// TIA Portal project "ProjectMurr-55510-en" (V18)

(* hardware
DEVICE "S7-1200 station_1"  S7-1200 Station
   slot 0: "Rack_0"  S7-1200 Rack  Rack  V1.0
   slot 1: "PLC_1"  CPU 1212FC DC/DC/DC  6ES7 212-1AF40-0XB0  V4.6
DEVICE "GSD device_1"  GSD.Device.PN
   slot 0: "Rack"  Rack  V1.0
   slot 0: "FIO"  FIO
   slot 0: "IOL_I/O_08/08 + PQI"  IOL_I/O_08/08 + PQI
   slot 0: "IOL_I/O_08/08 + PQI"  IOL_I/O_08/08 + PQI
   slot 0: "MVK-MPNIO-F"  55510 MVK PN FDI6/3 FDO2/1 DIO4 IOL2 IRT PP  55510  V1.03.00
      slot 0: "55510 MVK PN FDI6/3 FDO2/1 DIO4 IOL2 IRT PP_1"  55510 MVK PN FDI6/3 FDO2/1 DIO4 IOL2 IRT PP
      slot 1: "55510 MVK PN FDI6/3 FDO2/1 DIO4 IOL2 IRT PP"  55510 MVK PN FDI6/3 FDO2/1 DIO4 IOL2 IRT PP
         slot 1: "Port 1"  Port 1
         slot 2: "Port 2"  Port 2
      slot 1: "Device status_1"  Device status
         slot 0: "Parameters/Diagnostic"  Parameters/Diagnostic
   slot 2: "X0...X3 FDI/FDO_1"  X0...X3 FDI/FDO
   slot 3: "X4, X5 DIO_1"  X4, X5 DIO
      slot 0: "IOs, qualifier"  IOs, qualifier
   slot 4: "X6 IO-Link_1"  X6 IO-Link
      slot 1: "DI pin 2, qualifier"  DI pin 2, qualifier
   slot 5: "X7 IO-Link_1"  X7 IO-Link
*)

// ===== PLC "PLC_1"  CPU 1212FC DC/DC/DC =====

VAR_GLOBAL   // PLC tag table "Default tag table"
   "Murr_55510_SDI_S0" AT %I100.0 : "DUT_Murr_55510_SDI_b0";
   "Murr_55510_DSO" AT %Q100.0 : "DUT_Murr_55510_SDO_b0";
   "Murr_55510_IOLINK_Port6_IN" AT %I114.0 : "DUT_Nassmanget_SmartConnector_IN";
   "Murr_55510_IOLINK_Port7_IN" AT %I126.0 : "DUT_TURCKIOLU69X2_IN";
   "Murr_55510_IOLINK_Port6_OUT" AT %Q114.0 : "DUT_Nassmanget_SmartConnector_OUT";
   "Murr_5510_IOLINK_Port4_5_IN" AT %I110.0 : "DUT_Murr_55510_X4X5_PortBased_IN";
   "Murr_5510_IOLINK_Port4_5_OUT" AT %Q110.0 : "DUT_Murr_55510_X4X5_PortBased_OUT";
   "Murr_55510_SDI_S1_Q" AT %I101.0 : "DUT_Murr_55510_SDI_b0";
   "Murr_55510_SDI_S2" AT %I102.0 : "DUT_Murr_55510_SDI_b0";
END_VAR

TYPE "DUT_Murr_55510_SDI_b0"
   STRUCT
      FDI_X0_Pin4 : Bool;
      FDI_X1_Pin4 : Bool;
      FDI_X2_Pin4 : Bool;
      b3 : Bool;
      FDI_X0_Pin2 : Bool;
      FDI_X1_Pin2 : Bool;
      FDI_X2_Pin2 : Bool;
      b7 : Bool;
   END_STRUCT;
END_TYPE

TYPE "DUT_Murr_55510_SDI_b3"
   STRUCT
      FDO_X3_Pin4 : Bool;
      FDO_X3_Pin2 : Bool;
      FDO_X7_Pin2 : Bool;
      b3 : Bool;
      b4 : Bool;
      b5 : Bool;
      b6 : Bool;
      b7 : Bool;
   END_STRUCT;
END_TYPE

TYPE "DUT_Murr_55510_SDIs"
   STRUCT
      s0 : "DUT_Murr_55510_SDI_b0";
      s1_q : "DUT_Murr_55510_SDI_b0";
      s2 : "DUT_Murr_55510_SDI_b3";
   END_STRUCT;
END_TYPE

TYPE "DUT_Murr_55510_SDO_b0"
   STRUCT
      SDO_X3_Pin4 : Bool;
      SDO_X3_Pin2 : Bool;
      SDO_X7_Pin2 : Bool;
      b3 : Bool;
      b4 : Bool;
      b5 : Bool;
      b6 : Bool;
      b7 : Bool;
   END_STRUCT;
END_TYPE

TYPE "DUT_Murr_55510_SDOs"
   STRUCT
      s0 : "DUT_Murr_55510_SDO_b0";
   END_STRUCT;
END_TYPE

TYPE "DUT_Murr_55510_X4X5_Portbased_b0"
   STRUCT
      b0_X4_Pin4 : Bool;
      b1_X4_Pin2 : Bool;
      b2_X5_Pin4 : Bool;
      b3_X5_Pin2 : Bool;
      b4 : Bool;
      b5 : Bool;
      b6 : Bool;
      b7 : Bool;
   END_STRUCT;
END_TYPE

TYPE "DUT_Murr_55510_X4X5_PortBased_IN"
   STRUCT
      s0_DI : Byte;
      s1_DI_Q : Byte;
      s2_DO_Q : Byte;
   END_STRUCT;
END_TYPE

TYPE "DUT_Murr_55510_X4X5_PortBased_OUT"
   STRUCT
      S0_DO : "DUT_Murr_55510_X4X5_Portbased_b0";
   END_STRUCT;
END_TYPE

TYPE "DUT_Nassmanget_SmartConnector_IN"
   STRUCT
      b0_ValveState : Bool;
      b1_ShortCircuit : Bool;
      b2_OpenCircuit : Bool;
      b3_Overheat : Bool;
      b4_Overcurrent : Bool;
      b5_Counter1OverRun : Bool;
      b6_Counter2OverRun : Bool;
      b7 : Bool;
   END_STRUCT;
END_TYPE

TYPE "DUT_Nassmanget_SmartConnector_OUT"
   STRUCT
      b0_ONOFF : Bool;
      b1_PWM : Bool;
      b2_PWM : Bool;
      b3_PWM : Bool;
      b4_PWM : Bool;
      b5_PWM : Bool;
      b6_PWM : Bool;
      b7_PWM : Bool;
   END_STRUCT;
END_TYPE

TYPE "DUT_Nassmanget_SmartConnector_Data"
   STRUCT
      ValveState : Bool;
      ShortCircuit : Bool;
      OpenCircuit : Bool;
      Overheat : Bool;
      Overcurrent : Bool;
      Counter1OVerRun : Bool;
      Coutner2OverRun : Bool;
      ValveON : Bool;
      VlavePWM : Int;
   END_STRUCT;
END_TYPE

TYPE "DUT_TURCKIOLU69X2_IN"
   STRUCT
      b0_OutputState : Bool;
      b1_LowTemp_Warning : Bool;
      b2_HighTemp_Waring : Bool;
      b3_OutOfRange_Warning : Bool;
      b4_Analog : Bool;
      b5_Analog : Bool;
      b6_Analog : Bool;
      b7_Analog : Bool;
      b8_Analog : Bool;
      b9_Analog : Bool;
      b10_Analog : Bool;
      b11_Analog : Bool;
      b12_Analog : Bool;
      b13_Analog : Bool;
      b14_Analog : Bool;
      b15_Analog : Bool;
   END_STRUCT;
END_TYPE

TYPE "DUT_TURCKIOLU69X2_Data"
   STRUCT
      OutputState : Bool;
      LowTemp_Warning : Bool;
      HighTemp_Warning : Bool;
      OutOfRnage_Warning : Bool;
      AnalogValve : Real;
   END_STRUCT;
END_TYPE

DATA_BLOCK "Main_Safety_RTG1_DB"   // DB1, F_DB
{ S7_Optimized_Access := 'TRUE' }
NAME : FUSI
VERSION : 0.1
// stored: InstanceOfName Main_Safety_RTG1
"Main_Safety_RTG1"
BEGIN
END_DATA_BLOCK

DATA_BLOCK "DB_55510"   // DB2
{ S7_Optimized_Access := 'TRUE' }
VERSION : 0.1
   VAR
      Port7 : "DUT_TURCKIOLU69X2_Data";
      Port6 : "DUT_Nassmanget_SmartConnector_Data";
      Port5 : Struct
         iReset : Bool;
      END_STRUCT;
      Port4 : Struct
         qLamp : Bool;
      END_STRUCT;
   END_VAR
BEGIN
END_DATA_BLOCK

DATA_BLOCK "DB_SafetyExchange"   // DB3
{ S7_Optimized_Access := 'TRUE' }
VERSION : 0.1
   VAR
      ESTOP : Struct
         Q : Bool;
         Q_Delay : Bool;
         ACK_REQ : Bool;
         DIAG : Byte;
      END_STRUCT;
   END_VAR
BEGIN
END_DATA_BLOCK

DATA_BLOCK "FB_55510_DB"   // DB4
{ S7_Optimized_Access := 'TRUE' }
VERSION : 0.1
// stored: InstanceOfName FB_55510
"FB_55510"
BEGIN
END_DATA_BLOCK

FUNCTION_BLOCK "Main_Safety_RTG1"   // FB1, F_FBD
{ S7_Optimized_Access := 'TRUE' }
   VAR
      ESTOP1 : ESTOP1;
      ACK_GL_DB : ACK_GL;
   END_VAR
BEGIN

REGION Network 1
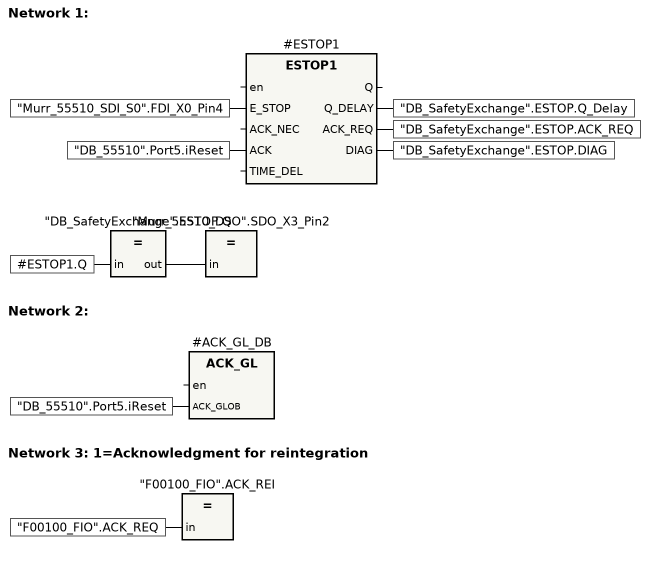
   #ESTOP1(E_STOP := "Murr_55510_SDI_S0".FDI_X0_Pin4,   // ESTOP1
           ACK := "DB_55510".Port5.iReset,
           Q_DELAY => "DB_SafetyExchange".ESTOP.Q_Delay,
           ACK_REQ => "DB_SafetyExchange".ESTOP.ACK_REQ,
           DIAG => "DB_SafetyExchange".ESTOP.DIAG);
   "DB_SafetyExchange".ESTOP.Q := #ESTOP1.Q;
   "Murr_55510_DSO".SDO_X3_Pin2 := #ESTOP1.Q;
END_REGION

REGION Network 2
   #ACK_GL_DB(ACK_GLOB := "DB_55510".Port5.iReset);   // ACK_GL
END_REGION

REGION Network 3: 1=Acknowledgment for reintegration
   "F00100_FIO".ACK_REI := "F00100_FIO".ACK_REQ;
END_REGION
END_FUNCTION_BLOCK

FUNCTION_BLOCK "FB_Nassmanget_SmartConnector"   // FB2, FBD
{ S7_Optimized_Access := 'TRUE' }
VERSION : 0.1
   VAR_IN_OUT
      rawIN : "DUT_Nassmanget_SmartConnector_IN";
      rawOut : "DUT_Nassmanget_SmartConnector_OUT";
      io : "DUT_Nassmanget_SmartConnector_Data";
   END_VAR
BEGIN

REGION Network 1
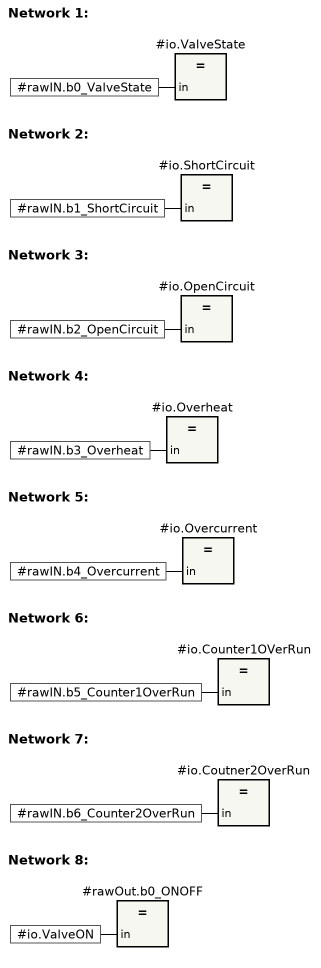
   #io.ValveState := #rawIN.b0_ValveState;
END_REGION

REGION Network 2
   #io.ShortCircuit := #rawIN.b1_ShortCircuit;
END_REGION

REGION Network 3
   #io.OpenCircuit := #rawIN.b2_OpenCircuit;
END_REGION

REGION Network 4
   #io.Overheat := #rawIN.b3_Overheat;
END_REGION

REGION Network 5
   #io.Overcurrent := #rawIN.b4_Overcurrent;
END_REGION

REGION Network 6
   #io.Counter1OVerRun := #rawIN.b5_Counter1OverRun;
END_REGION

REGION Network 7
   #io.Coutner2OverRun := #rawIN.b6_Counter2OverRun;
END_REGION

REGION Network 8
   #rawOut.b0_ONOFF := #io.ValveON;
END_REGION

REGION Network 9 (SCL)

   IF #io.VlavePWM < 0 OR #io.VlavePWM > 100 THEN

       #rawOut.b1_PWM := False;
       #rawOut.b2_PWM := False;
       #rawOut.b3_PWM := False;
       #rawOut.b4_PWM := False;
       #rawOut.b5_PWM := False;
       #rawOut.b6_PWM := False;
       #rawOut.b7_PWM := False;

   ELSE

       #rawOut.b1_PWM := #io.VlavePWM.%X0;
       #rawOut.b2_PWM := #io.VlavePWM.%X1;
       #rawOut.b3_PWM := #io.VlavePWM.%X2;
       #rawOut.b4_PWM := #io.VlavePWM.%X3;
       #rawOut.b5_PWM := #io.VlavePWM.%X4;
       #rawOut.b6_PWM := #io.VlavePWM.%X5;
       #rawOut.b7_PWM := #io.VlavePWM.%X6;



   END_IF;
END_REGION
END_FUNCTION_BLOCK

FUNCTION_BLOCK "FB_TURCKIOLU69X2"   // FB3, FBD
{ S7_Optimized_Access := 'TRUE' }
VERSION : 0.1
   VAR_IN_OUT
      rawIN : "DUT_TURCKIOLU69X2_IN";
      io : "DUT_TURCKIOLU69X2_Data";
   END_VAR
   VAR_TEMP
      _Temp : Int;
   END_VAR
BEGIN

REGION Network 1
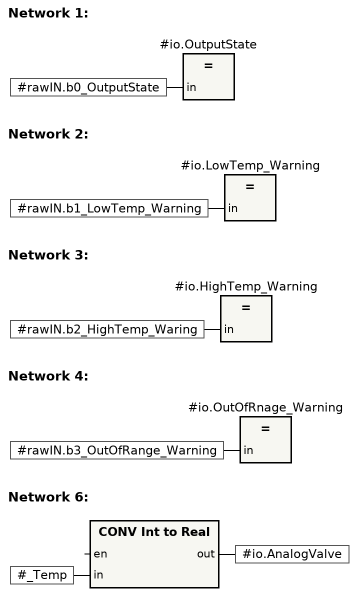
   #io.OutputState := #rawIN.b0_OutputState;
END_REGION

REGION Network 2
   #io.LowTemp_Warning := #rawIN.b1_LowTemp_Warning;
END_REGION

REGION Network 3
   #io.HighTemp_Warning := #rawIN.b2_HighTemp_Waring;
END_REGION

REGION Network 4
   #io.OutOfRnage_Warning := #rawIN.b3_OutOfRange_Warning;
END_REGION

REGION Network 5 (SCL)
   #_Temp.%X0 := #rawIN.b4_Analog;
   #_Temp.%X1 := #rawIN.b5_Analog;
   #_Temp.%X2 := #rawIN.b6_Analog;
   #_Temp.%X3 := #rawIN.b7_Analog;
   #_Temp.%X4 := #rawIN.b8_Analog;
   #_Temp.%X5 := #rawIN.b9_Analog;
   #_Temp.%X6 := #rawIN.b10_Analog;
   #_Temp.%X7 := #rawIN.b11_Analog;
   #_Temp.%X8 := #rawIN.b12_Analog;
   #_Temp.%X9 := #rawIN.b13_Analog;
   #_Temp.%X10 := #rawIN.b14_Analog;
   #_Temp.%X11 := #rawIN.b15_Analog;
END_REGION

REGION Network 6
   #io.AnalogValve := INT_TO_REAL(#_Temp);
END_REGION

REGION Network 7 (SCL)

   #io.AnalogValve :=
   ((#io.AnalogValve / 4095.0) * 3.0) + 0.2;
END_REGION
END_FUNCTION_BLOCK

FUNCTION_BLOCK "FB_55510"   // FB4, FBD
{ S7_Optimized_Access := 'TRUE' }
VERSION : 0.1
   VAR
      Port7 : "FB_TURCKIOLU69X2";
      Port6 : "FB_Nassmanget_SmartConnector";
      TON : TON_TIME;
   END_VAR
BEGIN

REGION Network 1
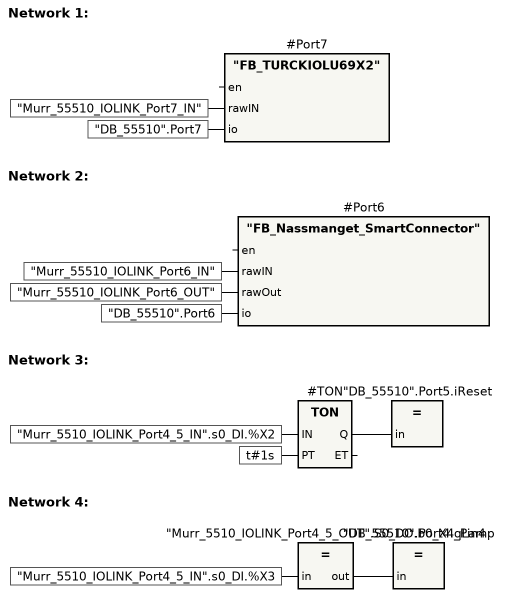
   #Port7(rawIN := "Murr_55510_IOLINK_Port7_IN", io := "DB_55510".Port7);   // "FB_TURCKIOLU69X2"
END_REGION

REGION Network 2
   #Port6(rawIN := "Murr_55510_IOLINK_Port6_IN",   // "FB_Nassmanget_SmartConnector"
          rawOut := "Murr_55510_IOLINK_Port6_OUT",
          io := "DB_55510".Port6);
END_REGION

REGION Network 3
   #TON(IN := "Murr_5510_IOLINK_Port4_5_IN".s0_DI.%X2, PT := t#1s);   // TON
   "DB_55510".Port5.iReset := #TON.Q;
END_REGION

REGION Network 4
   "Murr_5510_IOLINK_Port4_5_OUT".S0_DO.b0_X4_Pin4 := "Murr_5510_IOLINK_Port4_5_IN".s0_DI.%X3;
   "DB_55510".Port4.qLamp := "Murr_5510_IOLINK_Port4_5_IN".s0_DI.%X3;
END_REGION
END_FUNCTION_BLOCK

ORGANIZATION_BLOCK "Main"   // OB1, LAD, ProgramCycle
TITLE = "Main Program Sweep (Cycle)"
{ S7_Optimized_Access := 'TRUE' }
VERSION : 0.1
   VAR_INPUT
      Initial_Call : Bool;   // Initial call of this OB
      Remanence : Bool;   // =True, if remanent data are available
   END_VAR
BEGIN

REGION Network 1
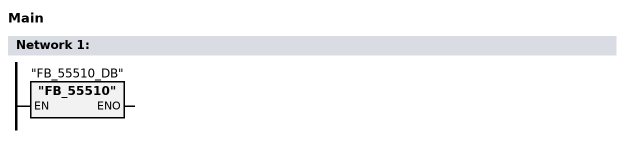
   RUNG wire#powerrail
      "FB_55510_DB"()
   END_RUNG
   // the same network as SCL:
   "FB_55510_DB"();   // "FB_55510"
END_REGION
END_ORGANIZATION_BLOCK